TYPE ST_Chamber1Ep1PrepardWaferTransferParam :
STRUCT
END_STRUCT
END_TYPE

(* stored: Version 1.1.0.1, ProductVersion 3.1.4026.18
   DUT ST_Chamber1Ep1PrepardWaferTransferParam: Id {b5a49ec2-cb1f-427e-897c-e69acfb39fec} *)
